{attribute 'GeneratedUsingTerminal: EL6910-0000-0017'}
{attribute addProperty BoxType "EL6910-0000-0017"}
{attribute addProperty Id "FSLOGIC_InputsAT %I*FSLOGIC_Inputs_EEE9388E2FSLOGIC_OutputsAT %I*EMPTY_STRUCTURE0WcStateAT %I*WcState_9091E0EB2InfoDataAT %I*InfoData_32EB74EA10"}
{attribute addProperty CRC "3444433408"}
{attribute addProperty Size "14"}
TYPE EL6910_CD4DE200 EXTENDS EtcSlaveTerminalBase_947E5A46 :
STRUCT
	{attribute addProperty Name "FSLOGIC_Inputs"}
	FSLOGIC_Inputs : FSLOGIC_Inputs_EEE9388E;
	{attribute addProperty Name "FSLOGIC_Outputs"}
	FSLOGIC_Outputs : EMPTY_STRUCTURE;
	{attribute addProperty Name "WcState"}
	WcState : WcState_9091E0EB;
	{attribute addProperty Name "InfoData"}
	InfoData : InfoData_32EB74EA;
END_STRUCT
END_TYPE

(* stored: Version 1.2.0.0, ProductVersion 3.1.4024.9
   DUT EL6910_CD4DE200: Id {aba9a7e1-6e04-4c2d-8f62-5beb74316550} *)
